{attribute addProperty BoxType "KL9528"}
{attribute addProperty Id "Channel_1Channel_53D9CDF100"}
{attribute addProperty CRC "1520347074"}
{attribute addProperty SizeInBites "0"}
{attribute addProperty SizeInBytes "0"}
TYPE KL9528_5A9EA7C2 :
STRUCT
	{attribute addProperty Name "Channel_1"}
	Channel_1 : Channel_53D9CDF1;
END_STRUCT
END_TYPE

(* stored: Version 1.2.0.0, ProductVersion 3.1.4024.9
   DUT KL9528_5A9EA7C2: Id {2d560413-16d1-401e-8a08-889cff489b6a} *)
